// TIA Portal V17 program export: 0 tag tables, 0 data types, 0 data blocks, 10 code blocks (in call order from the OBs), 2 instance data blocks

ORGANIZATION_BLOCK "Main"   // OB1, LAD, ProgramCycle
TITLE = "Main Program Sweep (Cycle)"
{ S7_Optimized_Access := 'TRUE' }
VERSION : 0.1
// stored: AutoNumber true, IsIECCheckEnabled false, SetENOAutomatically false
   VAR_INPUT
      Initial_Call : Bool;   // Initial call of this OB
      Remanence : Bool;   // =True, if remanent data are available
   END_VAR
BEGIN

REGION Network 1
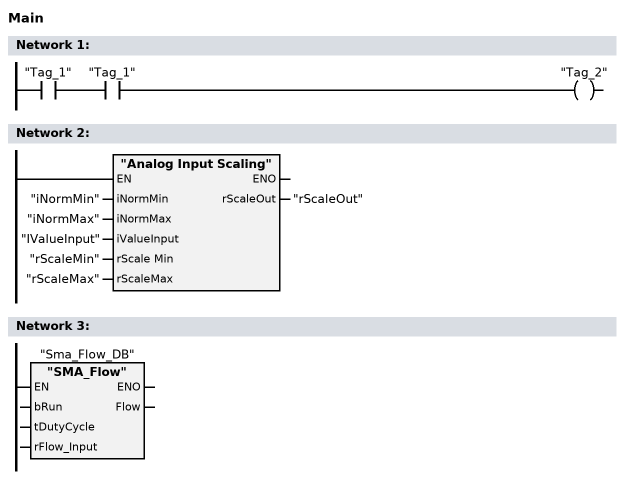
   RUNG wire#powerrail
      Contact( "Tag_1" )
      Contact( "Tag_1" )
      Coil( "Tag_2" )
   END_RUNG
   // the same network as SCL:
   "Tag_2" := "Tag_1" AND "Tag_1";
END_REGION

REGION Network 2
   RUNG wire#powerrail
      "Analog Input Scaling"(iNormMin := "iNormMin", iNormMax := "iNormMax", iValueInput := "IValueInput", "rScale Min" := "rScaleMin", rScaleMax := "rScaleMax", rScaleOut => "rScaleOut")
   END_RUNG
   // the same network as SCL:
   "Analog Input Scaling"(iNormMin := "iNormMin",
                          iNormMax := "iNormMax",
                          iValueInput := "IValueInput",
                          "rScale Min" := "rScaleMin",
                          rScaleMax := "rScaleMax",
                          rScaleOut => "rScaleOut");
END_REGION

REGION Network 3
   RUNG wire#powerrail
      "Sma_Flow_DB"(bRun :=, tDutyCycle :=, rFlow_Input :=, Flow =>)
   END_RUNG
   // the same network as SCL:
   "Sma_Flow_DB"();   // "SMA_Flow"
END_REGION
END_ORGANIZATION_BLOCK

FUNCTION "Analog Input Scaling" : Void   // FC2, LAD
{ S7_Optimized_Access := 'TRUE' }
VERSION : 0.1
// stored: AutoNumber true, IsIECCheckEnabled false, SetENOAutomatically false, UDAEnableTagReadback false
   VAR_INPUT
      iNormMin : Int;
      iNormMax : Int;
      iValueInput : Int;
      "rScale Min" : Real;
      rScaleMax : Real;
   END_VAR
   VAR_OUTPUT
      rScaleOut : Real;
   END_VAR
   VAR_TEMP
      rNormTemp : Real;
   END_VAR
BEGIN

REGION Network 1
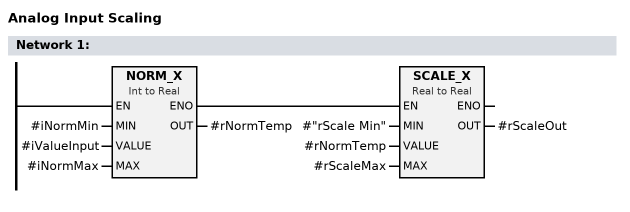
   RUNG wire#powerrail
      { S7_Templates := "[SrcType := Int, DestType := Real]" } Normalize(min := #iNormMin, value := #iValueInput, max := #iNormMax, out => #rNormTemp)
      { S7_Templates := "[SrcType := Real, DestType := Real]" } Scale(min := #"rScale Min", value := #rNormTemp, max := #rScaleMax, out => #rScaleOut)
   END_RUNG
   // the same network as SCL:
   #rNormTemp := NORM_X(MIN := #iNormMin, VALUE := #iValueInput, MAX := #iNormMax);
   #rScaleOut := SCALE_X(MIN := #"rScale Min", VALUE := #rNormTemp, MAX := #rScaleMax);
END_REGION
END_FUNCTION

FUNCTION_BLOCK "SMA_Flow"   // FB2, LAD
{ S7_Optimized_Access := 'TRUE' }
VERSION : 0.1
// stored: AutoNumber true, IsIECCheckEnabled false, IsRetainMemResEnabled false, MemoryReserve 100, SetENOAutomatically false, UDAEnableTagReadback false
   VAR_INPUT
      bRun : Bool;
      tDutyCycle : Time;
      rFlow_Input : Real;
   END_VAR
   VAR_OUTPUT
      Flow { ExternalAccessible := 'False'; ExternalVisible := 'False'; ExternalWritable := 'False'} : Real;
   END_VAR
   VAR_TEMP
      bCount : Bool;
      bpulse1 : Bool;
      iCount : Int;
      aFlow : Array[0..200] of Real;
      i : Int;
   END_VAR
   VAR_TEMP   // added for the SCL form of the ladder/FBD networks
      _w1 : Bool;
      _w2 : Bool;
   END_VAR
BEGIN

REGION Network 1
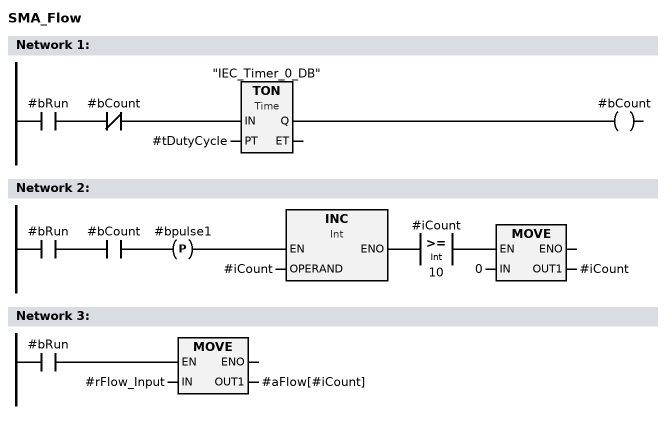
   RUNG wire#powerrail
      Contact( #bRun )
      I_Contact( #bCount )
      { S7_Templates := "time_type := Time" } "IEC_Timer_0_DB".TON(pt := #tDutyCycle, et =>)
      Coil( #bCount )
   END_RUNG
   // the same network as SCL:
   "IEC_Timer_0_DB".TON(IN := #bRun AND NOT #bCount, PT := #tDutyCycle);
   #bCount := "IEC_Timer_0_DB".Q;
END_REGION

REGION Network 2
   RUNG wire#powerrail
      Contact( #bRun )
      Contact( #bCount )
      P_Trig( #bpulse1 )
      { S7_Templates := "DestType := Int" } Inc( #iCount )
      { S7_Templates := "SrcType := Int" } GE_Contact(in1 := #iCount, in2 := 10)
      Move(in := 0, out1 => #iCount)
   END_RUNG
   // the same network as SCL:
   #_w1 := #bRun AND #bCount;
   #_w2 := #_w1 AND NOT #bpulse1;   // rising edge
   #bpulse1 := #_w1;
   IF #_w2 THEN #iCount := #iCount + 1; END_IF;
   IF #_w2 AND (#iCount >= 10) THEN #iCount := 0; END_IF;
END_REGION

REGION Network 3
   RUNG wire#powerrail
      Contact( #bRun )
      Move(in := #rFlow_Input, out1 => #aFlow[#iCount])
   END_RUNG
   // the same network as SCL:
   IF #bRun THEN #aFlow[#iCount] := #rFlow_Input; END_IF;
END_REGION

REGION Network 4 (SCL)
   FOR #i := 0 TO #iCount DO
       // Statement section FOR
       #Flow := #aFlow[#i] + #Flow;
       ;
   END_FOR;
END_REGION
END_FUNCTION_BLOCK

FUNCTION "Block_1" : Void   // FC1, LAD
{ S7_Optimized_Access := 'TRUE' }
VERSION : 0.1
// stored: AutoNumber true, IsIECCheckEnabled false, SetENOAutomatically false, UDAEnableTagReadback false
BEGIN
END_FUNCTION

FUNCTION_BLOCK "Counter & Pulse"   // FB3, LAD
{ S7_Optimized_Access := 'TRUE' }
VERSION : 0.1
// stored: AutoNumber true, IsIECCheckEnabled false, IsRetainMemResEnabled false, MemoryReserve 100, SetENOAutomatically false, UDAEnableTagReadback false
   VAR_INPUT
      bReset : Bool;
      bChangeHZ : Bool;
      bPuase : Bool;
   END_VAR
   VAR_OUTPUT
      iCvCounter : DInt;
   END_VAR
   VAR
      bCtu : Bool;
      bCtd : Bool;
   END_VAR
   VAR_TEMP   // added for the SCL form of the ladder/FBD networks
      _w1 : Bool;
   END_VAR
BEGIN

REGION Network 1
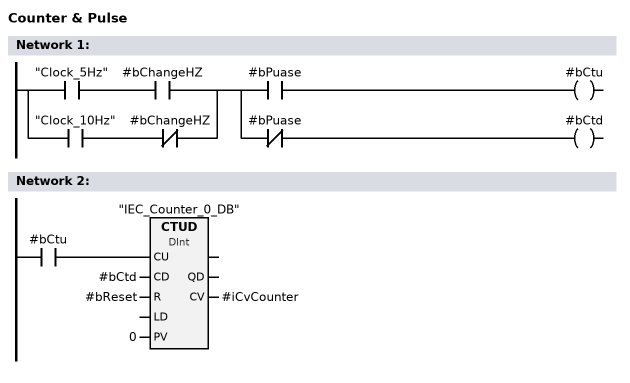
   RUNG wire#powerrail
      Contact( "Clock_5Hz" )
      Contact( #bChangeHZ )
      wire#w1
      Contact( #bPuase )
      Coil( #bCtu )
   END_RUNG
   RUNG wire#powerrail
      Contact( "Clock_10Hz" )
      I_Contact( #bChangeHZ )
   END_RUNG wire#w1
   RUNG wire#w1
      I_Contact( #bPuase )
      Coil( #bCtd )
   END_RUNG
   // the same network as SCL:
   #_w1 := ("Clock_5Hz" AND #bChangeHZ) OR ("Clock_10Hz" AND NOT #bChangeHZ);
   #bCtu := #_w1 AND #bPuase;
   #bCtd := #_w1 AND NOT #bPuase;
END_REGION

REGION Network 2
   RUNG wire#powerrail
      Contact( #bCtu )
      { S7_Templates := "value_type := DInt" } "IEC_Counter_0_DB".CTUD(cd := #bCtd, r := #bReset, ld :=, pv := 0, qd =>, cv => #iCvCounter)
   END_RUNG
   // the same network as SCL:
   "IEC_Counter_0_DB".CTUD(CU := #bCtu, CD := #bCtd, R := #bReset, PV := 0, CV => #iCvCounter);
END_REGION
END_FUNCTION_BLOCK

FUNCTION_BLOCK "Last version"   // FB6, LAD
{ S7_Optimized_Access := 'TRUE' }
VERSION : 0.1
// stored: AutoNumber true, IsIECCheckEnabled false, IsRetainMemResEnabled false, MemoryReserve 100, SetENOAutomatically false, UDAEnableTagReadback false
BEGIN

REGION Network 2: Calculate Flow
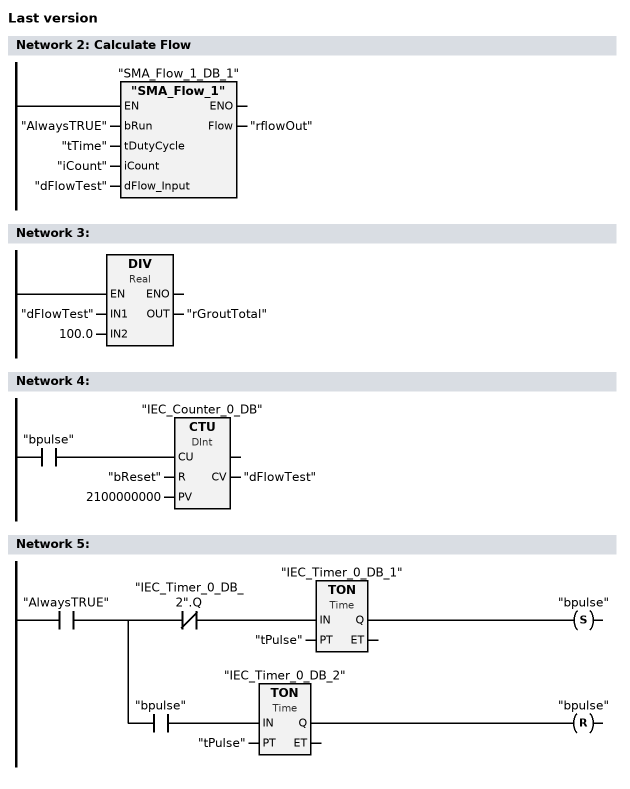
   RUNG wire#powerrail
      "SMA_Flow_1_DB_1"(bRun := "AlwaysTRUE", tDutyCycle := "tTime", iCount := "iCount", dFlow_Input := "dFlowTest", Flow => "rflowOut")
   END_RUNG
   // the same network as SCL:
   "SMA_Flow_1_DB_1"(bRun := "AlwaysTRUE",   // "SMA_Flow_1"
                     tDutyCycle := "tTime",
                     iCount := "iCount",
                     dFlow_Input := "dFlowTest",
                     Flow => "rflowOut");
END_REGION

REGION Network 3
   RUNG wire#powerrail
      { S7_Templates := "SrcType := Real" } Div(in1 := "dFlowTest", in2 := 100.0, out => "rGroutTotal")
   END_RUNG
   // the same network as SCL:
   "rGroutTotal" := "dFlowTest" / 100.0;
END_REGION

REGION Network 4
   RUNG wire#powerrail
      Contact( "bpulse" )
      { S7_Templates := "value_type := DInt" } "IEC_Counter_0_DB".CTU(r := "bReset", pv := 2100000000, cv => "dFlowTest")
   END_RUNG
   // the same network as SCL:
   "IEC_Counter_0_DB".CTU(CU := "bpulse", R := "bReset", PV := 2100000000, CV => "dFlowTest");
END_REGION

REGION Network 5
   RUNG wire#powerrail
      Contact( "AlwaysTRUE" )
      wire#w1
      I_Contact( "IEC_Timer_0_DB_2".Q )
      { S7_Templates := "time_type := Time" } "IEC_Timer_0_DB_1".TON(pt := "tPulse", et =>)
      S_Coil( "bpulse" )
   END_RUNG
   RUNG wire#w1
      Contact( "bpulse" )
      { S7_Templates := "time_type := Time" } "IEC_Timer_0_DB_2".TON(pt := "tPulse", et =>)
      R_Coil( "bpulse" )
   END_RUNG
   // the same network as SCL:
   "IEC_Timer_0_DB_1".TON(IN := "AlwaysTRUE" AND NOT "IEC_Timer_0_DB_2".Q, PT := "tPulse");
   IF "IEC_Timer_0_DB_1".Q THEN "bpulse" := TRUE; END_IF;
   "IEC_Timer_0_DB_2".TON(IN := "AlwaysTRUE" AND "bpulse", PT := "tPulse");
   IF "IEC_Timer_0_DB_2".Q THEN "bpulse" := FALSE; END_IF;
END_REGION

REGION Network 6: Start ReCording...
END_REGION
END_FUNCTION_BLOCK

FUNCTION_BLOCK "SMA_Flow_1"   // FB2, LAD
{ S7_Optimized_Access := 'TRUE' }
VERSION : 0.1
// stored: AutoNumber true, IsIECCheckEnabled false, IsRetainMemResEnabled false, MemoryReserve 100, SetENOAutomatically false, UDAEnableTagReadback false
   VAR_INPUT
      bRun : Bool;
      tDutyCycle : Time;
      rFlow_Input : Real;
   END_VAR
   VAR_OUTPUT
      Flow { ExternalAccessible := 'False'; ExternalVisible := 'False'; ExternalWritable := 'False'} : Real;
   END_VAR
   VAR_TEMP
      bCount : Bool;
      bpulse1 : Bool;
      iCount : Int;
      aFlow : Array[0..200] of Real;
      i : Int;
   END_VAR
   VAR_TEMP   // added for the SCL form of the ladder/FBD networks
      _w1 : Bool;
      _w2 : Bool;
   END_VAR
BEGIN

REGION Network 1
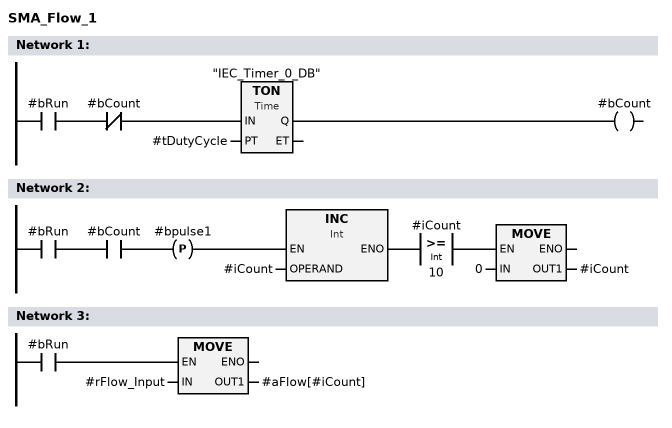
   RUNG wire#powerrail
      Contact( #bRun )
      I_Contact( #bCount )
      { S7_Templates := "time_type := Time" } "IEC_Timer_0_DB".TON(pt := #tDutyCycle, et =>)
      Coil( #bCount )
   END_RUNG
   // the same network as SCL:
   "IEC_Timer_0_DB".TON(IN := #bRun AND NOT #bCount, PT := #tDutyCycle);
   #bCount := "IEC_Timer_0_DB".Q;
END_REGION

REGION Network 2
   RUNG wire#powerrail
      Contact( #bRun )
      Contact( #bCount )
      P_Trig( #bpulse1 )
      { S7_Templates := "DestType := Int" } Inc( #iCount )
      { S7_Templates := "SrcType := Int" } GE_Contact(in1 := #iCount, in2 := 10)
      Move(in := 0, out1 => #iCount)
   END_RUNG
   // the same network as SCL:
   #_w1 := #bRun AND #bCount;
   #_w2 := #_w1 AND NOT #bpulse1;   // rising edge
   #bpulse1 := #_w1;
   IF #_w2 THEN #iCount := #iCount + 1; END_IF;
   IF #_w2 AND (#iCount >= 10) THEN #iCount := 0; END_IF;
END_REGION

REGION Network 3
   RUNG wire#powerrail
      Contact( #bRun )
      Move(in := #rFlow_Input, out1 => #aFlow[#iCount])
   END_RUNG
   // the same network as SCL:
   IF #bRun THEN #aFlow[#iCount] := #rFlow_Input; END_IF;
END_REGION

REGION Network 4 (SCL)
   FOR #i := 0 TO #iCount DO
       // Statement section FOR
       #Flow := #aFlow[#i] + #Flow;
       ;
   END_FOR;
END_REGION
END_FUNCTION_BLOCK

FUNCTION_BLOCK "Move Average Test"   // FB5, LAD
{ S7_Optimized_Access := 'TRUE' }
VERSION : 0.1
// stored: AutoNumber true, IsIECCheckEnabled false, IsRetainMemResEnabled false, MemoryReserve 100, SetENOAutomatically false, UDAEnableTagReadback false
   VAR_TEMP   // added for the SCL form of the ladder/FBD networks
      _w1 : Bool;
   END_VAR
BEGIN

REGION Network 1
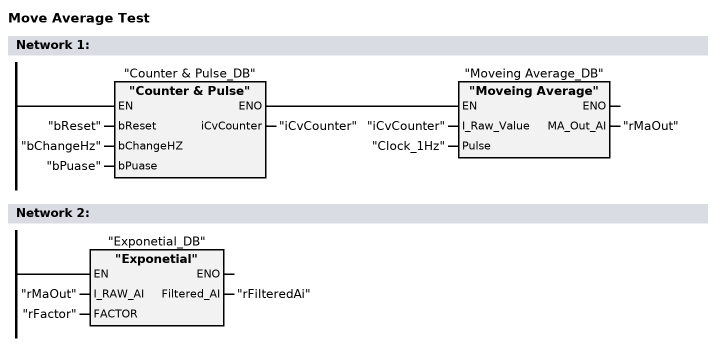
   RUNG wire#powerrail
      "Counter & Pulse_DB"(bReset := "bReset", bChangeHZ := "bChangeHz", bPuase := "bPuase", iCvCounter => "iCvCounter")
      "Moveing Average_DB"(I_Raw_Value := "iCvCounter", Pulse := "Clock_1Hz", MA_Out_AI => "rMaOut")
   END_RUNG
   // the same network as SCL:
   "Counter & Pulse_DB"(bReset := "bReset",   // "Counter & Pulse"
                        bChangeHZ := "bChangeHz",
                        bPuase := "bPuase",
                        iCvCounter => "iCvCounter",
                        ENO => #_w1);
   IF #_w1 THEN
       "Moveing Average_DB"(I_Raw_Value := "iCvCounter", Pulse := "Clock_1Hz", MA_Out_AI => "rMaOut");   // "Moveing Average"
   END_IF;
END_REGION

REGION Network 2
   RUNG wire#powerrail
      "Exponetial_DB"(I_RAW_AI := "rMaOut", FACTOR := "rFactor", Filtered_AI => "rFilteredAi")
   END_RUNG
   // the same network as SCL:
   "Exponetial_DB"(I_RAW_AI := "rMaOut", FACTOR := "rFactor", Filtered_AI => "rFilteredAi");   // "Exponetial"
END_REGION
END_FUNCTION_BLOCK

FUNCTION_BLOCK "Moveing Average"
{ S7_Optimized_Access := 'TRUE' }
VERSION : 0.1
   VAR_INPUT 
      I_Raw_Value : Real;
      Pulse : Bool;
   END_VAR

   VAR_OUTPUT 
      MA_Out_AI : Real;
   END_VAR

   VAR 
      Average : Real;
      Sum : Real;
      i : Int;
      StatePulse : Bool;
      StateFlag : Bool := false;
      StateEdge : Bool := false;
      Buffer : Array[0..#PERIOD] of Real;
   END_VAR

   VAR CONSTANT 
      PERIOD : Int := 5;
   END_VAR


BEGIN
	
	
	IF #i > #PERIOD - 1 THEN
	    #i := 0;
	    
	END_IF;
	
	IF #i < 0 THEN
	    #i := 0;
	    ;
	END_IF;
	
	#StatePulse := #Pulse;
	
	#StateEdge := #StatePulse AND NOT #StateFlag;
	#StateFlag := #StatePulse;
	
	IF (#StateEdge) THEN
	    
	    #Sum := #Sum + #I_Raw_Value - #Buffer[#i];
	    #Buffer[#i] := #I_Raw_Value;
	    #i := #i + 1;
	    #Average := #Sum / #PERIOD;
	    #MA_Out_AI := #Average;
	    
	END_IF;
END_FUNCTION_BLOCK

FUNCTION_BLOCK "Exponetial"
{ S7_Optimized_Access := 'TRUE' }
VERSION : 0.1
   VAR_INPUT 
      I_RAW_AI : Real;
      FACTOR : Real;
   END_VAR

   VAR_OUTPUT 
      Filtered_AI : Real;
   END_VAR

   VAR 
      Static_FILTERED_AI : Real;
   END_VAR


BEGIN
	#Static_FILTERED_AI := #FACTOR * #I_RAW_AI + (1 - #FACTOR) * #Static_FILTERED_AI;
	#Filtered_AI := #Static_FILTERED_AI;
	
END_FUNCTION_BLOCK

DATA_BLOCK "SMA_Flow_1_DB"   // DB5
VERSION : 0.1
// stored: AutoNumber true, DBAccessibleFromOPCUA true, InstanceOfName SMA_Flow_1, InstanceOfType FB
"SMA_Flow_1"
BEGIN
END_DATA_BLOCK

DATA_BLOCK "Sma_Flow_DB"   // DB4
VERSION : 0.1
// stored: AutoNumber true, DBAccessibleFromOPCUA true, InstanceOfName Sma_Flow, InstanceOfType FB
"Sma_Flow"
BEGIN
END_DATA_BLOCK
